// TwinCAT 3 PLC project PlcProject2
// ProgramVersion: 3.1.4023.0
// libraries:
//   Tc2_Standard, * (Beckhoff Automation GmbH)
//   Tc2_System, * (Beckhoff Automation GmbH)
//   Tc3_Module, * (Beckhoff Automation GmbH)
//   TcUnit, * (www.tcunit.org)
// project tree:
//   / PlcTask.TcTTO
//   POUs/ MAIN.TcPOU
// (motion and I/O tree: see PLC project plcproject1)
// real-time tasks:
//   TASK PlcTask: cycle T#10ms, priority 20, ADS port 350
//   TASK PlcTask1: cycle T#10ms, priority 21, ADS port 351

CONFIGURATION PlcProject2
    RESOURCE PLC ON TwinCAT3
        TASK PlcTask(INTERVAL := T#10ms, PRIORITY := 21);
        PROGRAM MAIN WITH PlcTask : MAIN;
    END_RESOURCE
END_CONFIGURATION

// ---- POUs/MAIN.TcPOU
PROGRAM MAIN
VAR
	bToggle : BOOL;
	bArray	: ARRAY[0..1] OF BOOL;
	f1 : LREAL := 10;
	f2 : LREAL := 1.0;
	idx : INT := 0;
END_VAR


bToggle := NOT bToggle;
f2 := 1;

//f1 := f1 / f2;

(*
FOR idx := -1 TO 2 DO
	bArray[idx] := bToggle;
END_FOR;
*)

END_PROGRAM
